Staubli VAL3: checkMotStack.pgx

program checkMotStack()
begin
  //!brief
  //This routine sets a warnig if the motion stack has been empty for more than WAR_MOTIONSTACK seconds.

  if (clock()-tmMotionStack>WAR_MOTIONSTACK) and !bDisplayed and isEmpty()
    ///TODO
    //call status:raise()
    //call ui:popUp((("The routine StartMachine() was called, but the arm is not programmed to leave the mould!")),data:nMsgTimeOut,false)
    bDisplayed=true
  endIf
end
